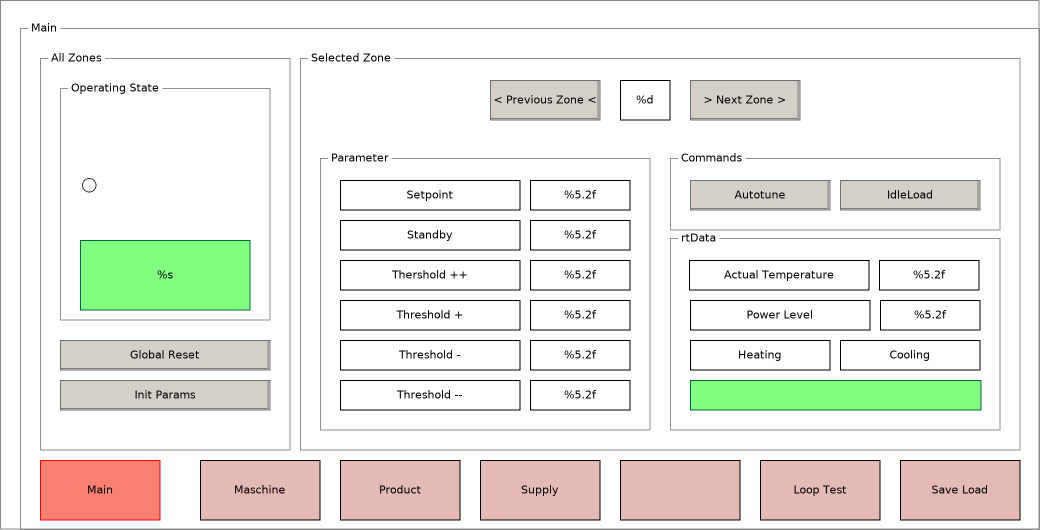
VISUALIZATION Visu_Main  // 1040x530
    GroupBox (20,20 1020x510), "Main"
        Rectangle (20,440 120x60), "Main"
            OnMouseClick: change screen: Visu_Main
        Rectangle (880,440 120x60), "Save Load"
            OnMouseClick: change screen: Visu_SaveLoad
        Rectangle (320,440 120x60), "Product"
            OnMouseClick: change screen: Visu_PParam
        Rectangle (180,440 120x60), "Maschine"
            OnMouseClick: change screen: Visu_MParam
    GroupBox (40,50 250x400), "All Zones", input disabled if: TemperatureCtrl.eState<>eMainSM_Idle
        GroupBox (20,30 210x240), "Operating State", input disabled if: TemperatureCtrl.eState<>eMainSM_Idle
            RadioButton (20,30 150x150), variable: eStatus
                Areas[0]: Text=Off
                Areas[1]: Text=Standby
                Areas[2]: Text=On
                Areas[3]: Text=Autotune
                Areas[4]: Text=Idle Load
            Rectangle (20,160 170x70), "%s", text variable: sErrorText, colour toggle: bGlobalError
        Button (20,330 210x30), "Init Params"
            tap bParamsInit
        Button (20,290 210x30), "Global Reset"
            tap aaaTempFault_Reset
    GroupBox (300,50 720x400), "Selected Zone"
        Rectangle (320,30 50x40), "%d", text variable: nVisuCount
        Button (190,30 110x40), "< Previous Zone <"
            tap bVisuBefore
        Button (390,30 110x40), "> Next Zone >"
            tap bVisuNext
        GroupBox (20,100 330x280), "Parameter"
            Rectangle (20,30 180x30), "Setpoint"
            Rectangle (20,70 180x30), "Standby"
            Rectangle (20,110 180x30), "Thershold ++"
            Rectangle (20,150 180x30), "Threshold +"
            Rectangle (20,190 180x30), "Threshold -"
            Rectangle (20,230 180x30), "Threshold --"
            Rectangle (210,30 100x30), "%5.2f", text variable: aaaPfwTempPparamFromHmi[nVisuCount].Setpoint
            Rectangle (210,70 100x30), "%5.2f", text variable: aaaPfwTempPparamFromHmi[nVisuCount].StandbySetpoint
            Rectangle (210,110 100x30), "%5.2f", text variable: aaaPfwTempPparamFromHmi[nVisuCount].Threshold_PP
            Rectangle (210,150 100x30), "%5.2f", text variable: aaaPfwTempPparamFromHmi[nVisuCount].Threshold_P
            Rectangle (210,190 100x30), "%5.2f", text variable: aaaPfwTempPparamFromHmi[nVisuCount].Threshold_M
            Rectangle (210,230 100x30), "%5.2f", text variable: aaaPfwTempPparamFromHmi[nVisuCount].Threshold_MM
        GroupBox (370,180 330x200), "rtData"
            Rectangle (210,70 100x30), "%5.2f", text variable: aaaPfwTempToHmi[nVisuCount].PowerLevel
            Rectangle (19,30 180x30), "Actual Temperature"
            Rectangle (209,30 100x30), "%5.2f", text variable: aaaPfwTempToHmi[nVisuCount].ActualTemp
            Rectangle (20,70 180x30), "Power Level"
            Rectangle (170,110 140x30), "Cooling", colour toggle: aaaPfwTempToHmi[nVisuCount].Cooling
            Rectangle (20,110 140x30), "Heating", colour toggle: aaaPfwTempToHmi[nVisuCount].Heating
            Rectangle (20,150 291x30), colour toggle: aaaPfwTempToHmi[nVisuCount].Error, text list: 'TL_TcPfw_ErrorId', text index: INT_TO_STRING(aaaPfwTempToHmi[nVisuCount].ErrorId)
                OnMouseClick: ChangeLanguage ChangeLanguage=en
        GroupBox (370,100 330x80), "Commands", input disabled if: aaaPfwTempMparamFromHmi[nVisuCount].Autotune OR aaaPfwTempMparamFromHmi[nVisuCount].Ena_TuneIdleLoad OR TemperatureCtrl.eState<>eMainSM_Idle
            Button (20,30 140x30), "Autotune"
                tap bVisuAutotune
            Button (170,30 140x30), "IdleLoad"
                tap bVisuIdleLoad
    Rectangle (480,460 120x60), "Supply"
        OnMouseClick: change screen: Visu_Supply
    Rectangle (620,460 120x60)
    Rectangle (760,460 120x60), "Loop Test"
        OnMouseClick: change screen: Visu_LoopTest
END_VISUALIZATION

(* stored: Version 1.1.0.1
   Visu Visu_Main: Id {7b811d24-4c30-4186-9ff1-bcae1788ca85} *)
